FUNCTION_BLOCK FB_Flasher
VAR
	timON: TON;
	timOFF: TON;
END_VAR

VAR_INPUT
	timeVal:TIME;
	
END_VAR

VAR_OUTPUT
	q:BOOL;

END_VAR

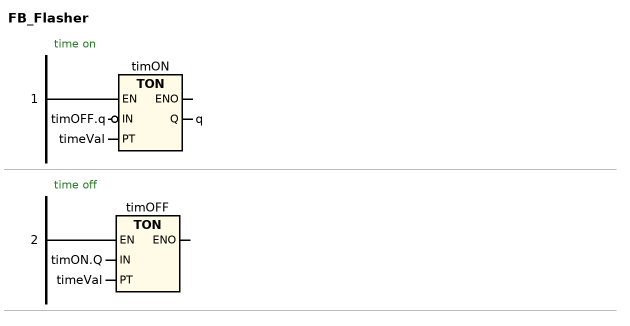
// NETWORK 1
// time on
timON(IN := NOT timOFF.q, PT := timeVal, Q => q); // TON

// NETWORK 2
// time off
timOFF(IN := timON.Q, PT := timeVal); // TON

END_FUNCTION_BLOCK

(* stored: Version 1.1.0.1, ProductVersion 3.1.4024.12
   POU FB_Flasher: Id {ab9ee524-2100-4c00-9352-d5c1d062606f}, SpecialFunc None *)
